// TIA Portal V20 export
// export: Created 2025-12-01T14:57:10.651905Z, ExportSetting None, DisplayName Totally Integrated Automation Portal, DisplayVersion V20 Update 3, DisplayName TIA Portal Openness, DisplayVersion V20 Update 3, DisplayName TIA Portal Version Control Interface, DisplayVersion V20 Update 3, DisplayName STEP 7 Professional, DisplayVersion V20 Update 3, DisplayName STEP 7 Safety, DisplayVersion V20 Update 2, DisplayName WinCC Basic/Comfort/Advanced, DisplayVersion V20 Update 3, DisplayName WinCC Professional, DisplayVersion V20 Update 3, DisplayName WinCC Unified, DisplayVersion V20 Update 3
FUNCTION "FC822_EstadosMesas" : Void   // FC822, LAD
TITLE = "EstadosMesas" - Calcular los eventos con las Mesas
{ S7_Optimized_Access := 'FALSE' }
AUTHOR : TRACKING
NAME : 20170706
VERSION : 4.6
// - Inicializaciones
// - Bucle de Mesas
// - Cierre de protocolo
// - Calculo de los Eventos con Presencias
// - Calculo de los Eventos Generales
// stored: AutoNumber false, SetENOAutomatically false
   VAR_TEMP
      EmiProtocoloDeMesa : "UDT_ProtocoloEmiMesa";
      P_EmiProtocolo : DWord;
      NumeroMesa : UInt;   // Numero de Mesa Actual
      NumeroUT : UInt;   // Numero de UT Actual
      SiguienteUT : UInt;   // Numero de UT Siguiente
      AnteriorUT : UInt;
      GaliboTMP : Word;
      HuecoTacoTMP : Word;
      AlturaTMP : UInt;
      ValorTMP : UInt;
      GrupoTMP : UInt;
   END_VAR
BEGIN

NETWORK
TITLE = Inicializar
// - Inicializacion de las variables de los DB's
/////////////////////////////////////////////////////////////////////////
// --- Inicializaciones de las variables de los DB's



NETWORK
TITLE = Bucle de Mesas
// - Inicializacion de los punteros de la mesa (PunteroMesa y PunteroPLC)
// - Inicializacion de la definicion de la Mesa
// - Mirar si ha cerrado el protocolo
// - Mirar si hay UT's en la Mesa
// -
/////////////////////////////////////////////////////////////////////////
//                      Recorrer todas las Mesas
/////////////////////////////////////////////////////////////////////////
// -- Inicializacion de los Punteros de la Mesa
// -- Miarar si ha cerrado el protocolo de la Mesa

      L     0;  // Inicializo variable, para bucle de mesas
      T     #NumeroMesa;

/////////////////////////////////////////////////////////////////////////
// --- Empieza el recorrido por todas las Mesas
InicioBucle_Mesas:NOP   0;
      L     #NumeroMesa;  // Incremento en uno el numero de mesa
      L     1;
      +I;
      T     #NumeroMesa;


/////////////////////////////////////////////////////////////////////////
// Ya estan todas las Mesas
      L     #NumeroMesa;
      L     "CTE_MaxMesas";
      >I;
      JC    _END;  // Ya he recorrido todas las Mesas


/////////////////////////////////////////////////////////////////////////
/// Mirar Si hay Mesa Configurada

      SET;
      AN    "DB850_DefinicionMesas".Mesa[#NumeroMesa].ConfigMesa.MesaPaso;
      AN    "DB850_DefinicionMesas".Mesa[#NumeroMesa].ConfigMesa.MesaCruce;
      AN    "DB850_DefinicionMesas".Mesa[#NumeroMesa].ConfigMesa.MesaMultiplesDestinos;
      AN    "DB850_DefinicionMesas".Mesa[#NumeroMesa].ConfigMesa.MesaTL;
      JC    InicioBucle_Mesas;


/////////////////////////////////////////////////////////////////////////
/// Recoger Datos de Emision y Recepcion
// --- Recoger Datos del Dispositivo (Protocolo)
      CALL  MOVE
      ( IN  := "DB840_Emision".Mesa[#NumeroMesa].Protocolo,
        OUT := #EmiProtocoloDeMesa
      );

      L     P##EmiProtocoloDeMesa;
      T     #P_EmiProtocolo;


/////////////////////////////////////////////////////////////////////////
// --- Mirar si ha cerrado el protocolo de la Mesa

      L     "DB810_ColasMesas".Colas[#NumeroMesa].EstadoPresenciaMesa;
      L     0;  // Mirar si no esta Cerrado el Protocolo
      <>I;  // Ir a Cerrar Protocolo de la Mesa
      JC    CerrarProtocolo_Mesa;


/////////////////////////////////////////////////////////////////////////
// --- Mirar si hay UT's en la Mesa
//     Mirar si existe una UT, coger la primera
      L     "DB810_ColasMesas".Colas[#NumeroMesa].UT_PrimeraMesa;
      T     #NumeroUT;  // UT_Primera

      L     #NumeroUT;
      L     0;
      ==I;
      JC    InicioBucle_Mesas;  // No hay UT's en la Mesa, Siguiente Mesa


/////////////////////////////////////////////////////////////////////////
// --- Tratar la Mesa
      JU    TratarPresencias_Mesa;



NETWORK
TITLE = Cierre del protocolo de la mesa
// - Recoger como esta la Presencia
// - Distribuir dependiendo del Status del Protocolo
//   * Esta en Fase 1 - Esperando que se desactive la Presencia de la Mesa
CerrarProtocolo_Mesa:NOP   0;

/////////////////////////////////////////////////////////////////////////
/////////////////////////////////////////////////////////////////////////
/////////////////////////////////////////////////////////////////////////
/////////////////////////////////////////////////////////////////////////
// --- Mirar si ha desactivado todas las presencias
      L     LW [#P_EmiProtocolo];
      L     W#16#FF7F;
      AW;
      L     0;
      <>I;  // Estan Desactivados ?
      JC    FinCerrarProtocolo_Mesa;


/////////////////////////////////////////////////////////////////////////
// --- Fase 1 - Esperando que se desactive Emision de la Mesa
      SET;  // DesActivar - EmiOK de la Mesa
      R     "DB841_Recepcion".Mesa[#NumeroMesa].Protocolo.EmiOK;

      L     0;  // Fase 0 - Acabado el Protocolo
      T     "DB810_ColasMesas".Colas[#NumeroMesa].EstadoPresenciaMesa;


/////////////////////////////////////////////////////////////////////////
// --- Final del Segmento del Cierre de Protocolo de la Mesa
FinCerrarProtocolo_Mesa:NOP   0;
// Finalizar, Siguiente Mesa
      JU    InicioBucle_Mesas;



NETWORK
TITLE = Empezar el cierre del protocolo
// Empezar el cierre del protocolo - Empezar el EmiOK
EmpezarProtocolo_Mesa:NOP   0;

/////////////////////////////////////////////////////////////////////////
/////////////////////////////////////////////////////////////////////////
/////////////////////////////////////////////////////////////////////////
/////////////////////////////////////////////////////////////////////////
// --- Empezar el cierre del protocolo
      SET;  // Activar - EmiOK de la Mesa
      S     "DB841_Recepcion".Mesa[#NumeroMesa].Protocolo.EmiOK;

      L     1;  // Fase 1, Empezar el Protocolo
      T     "DB810_ColasMesas".Colas[#NumeroMesa].EstadoPresenciaMesa;


/////////////////////////////////////////////////////////////////////////
// Finalizar, Siguiente Mesa
      JU    InicioBucle_Mesas;



NETWORK
TITLE = Tratamiento de la Mesa
// - Tratamiento de la presencia de una mesa
//   * Leer del PLC la Zona de Bits
//   * Miramos si hay alguno activo
//     * Si hay alguno: Distribucion del Tipo de Presencias
//     * Si no hay alguno: Vamos a Generales
TratarPresencias_Mesa:NOP   0;

/////////////////////////////////////////////////////////////////////////
/////////////////////////////////////////////////////////////////////////
/////////////////////////////////////////////////////////////////////////
// --- Miramos si hay alguno activo

      L     LW [#P_EmiProtocolo];  // Zona de Bits
      L     W#16#FF7F;  // Quitamos el bit RecepOK
      AW;
      L     0;  // Mirar si hay alguno activo
      ==I;  // Ir a tratar Estado General
      JC    TratarEstadoGeneral_Mesa;

/////////////////////////////////////////////////////////////////////////
/////////////////////////////////////////////////////////////////////////
// --- Distribuir dependiendo del tipo de presencia

/////////////////////////////////////////////////////////////////////////
// Evento de Presencia Normal
      SET;  // Al final de la Cola
      A     #EmiProtocoloDeMesa.PresNormal;
      AN    #EmiProtocoloDeMesa.PresReset;
      AN    "DB850_DefinicionMesas".Mesa[#NumeroMesa].ConfigMesa.MeterAlPrincipio;
      JC    TratarPresenciaUltimaUT_Mesa;

      SET;  // Al principio de la Cola
      A     #EmiProtocoloDeMesa.PresNormal;
      AN    #EmiProtocoloDeMesa.PresReset;
      A     "DB850_DefinicionMesas".Mesa[#NumeroMesa].ConfigMesa.MeterAlPrincipio;
      JC    TratarPresenciaPrimeraUT_Mesa;

/////////////////////////////////////////////////////////////////////////
// Evento de Presencia con Galibo
      SET;  // Al final de la Cola
      A     #EmiProtocoloDeMesa.PresGalibo;
      AN    "DB850_DefinicionMesas".Mesa[#NumeroMesa].ConfigMesa.MeterAlPrincipio;
      JC    TratarGaliboUltimaUT_Mesa;

      SET;  // Al principio de la Cola
      A     #EmiProtocoloDeMesa.PresGalibo;
      A     "DB850_DefinicionMesas".Mesa[#NumeroMesa].ConfigMesa.MeterAlPrincipio;
      JC    TratarGaliboPrimeraUT_Mesa;

/////////////////////////////////////////////////////////////////////////
// Evento de Presencia con Bloqueo
      SET;
      A     #EmiProtocoloDeMesa.PresBloqueo;
      JC    TratarPresenciaBloqueo_Mesa;

/////////////////////////////////////////////////////////////////////////
// Evento de Presencia de Reset
      SET;
      A     #EmiProtocoloDeMesa.PresNormal;
      A     #EmiProtocoloDeMesa.PresReset;
      JC    TratarPresenciaReset_Mesa;

/////////////////////////////////////////////////////////////////////////
// Evento de Ausencia
      SET;  // (BORRAR UT)
      A     "DB850_DefinicionMesas".Mesa[#NumeroMesa].ConfigMesa.AusenciaBorrarUT;
      A     #EmiProtocoloDeMesa.Ausencia;
      JC    TratarAusenciaBorrar_Mesa;

      SET;  // (NORMAL)
      AN    "DB850_DefinicionMesas".Mesa[#NumeroMesa].ConfigMesa.AusenciaBorrarUT;
      A     #EmiProtocoloDeMesa.Ausencia;
      JC    TratarAusenciaNormal_Mesa;


/////////////////////////////////////////////////////////////////////////
// --- Si llega aqui este tipo no esta programado
// Ir a Empezar el Cierre de Protocolo
      JU    CerrarProtocolo_Mesa;



NETWORK
TITLE = Tratamiento de los Eventos Generales
// - Recorrer todas las UT's de la Mesa
//   - Recoger datos de la UT
//   - Mirar si se pueden generar eventos
//     * StatusEventoAGenerar = 0
//     * StatusEmision = 0
//     * StatusRecepcion = 0
//   - Mirar si tiene eventos generales
//     * Evento de Peticion de ruta 
//     * Evento de Refesco de datos
//     * Evento de Peticion de datos
//     * Nueva UT en Mesa (No se debe dar nunca)
//     * Borrar UT
// - Siguiente UT (Si hay más en la Mesa)
TratarEstadoGeneral_Mesa:NOP   0;

/////////////////////////////////////////////////////////////////////////
/////////////////////////////////////////////////////////////////////////
/////////////////////////////////////////////////////////////////////////
// --- Recorrer todas las Ut's de la Mesa
InicioBucleUTs_Mesa:NOP   0;

/////////////////////////////////////////////////////////////////////////
// --- Mirar si de pueden Generar eventos
//     - Si hay algo para generar
//     - Si puede ?

// --- No hay nada que generar
      L     "DB812_UTs_Control".UT[#NumeroUT].EstadoGeneralUT;
      L     0;  // EstaodGeneralUT <> 0
      ==I;  // Siguiente UT de la Mesa, No hay
      JC    ContinuarBucleUTs_Mesa;

// --- Se puede ?
      L     "DB812_UTs_Control".UT[#NumeroUT].EstadoEventoAGenerar;
      L     0;  // EstaodEventoAGenerar = 0
      <>I;  // Siguiente UT de la Mesa, No se puede
      JC    ContinuarBucleUTs_Mesa;

// --- Siempre se Borra UT
//     Evento de BorrarUT
      L     "DB812_UTs_Control".UT[#NumeroUT].EstadoGeneralUT;
      L     31;  // 31 - Borrar UT
      ==I;  // No hay cumplir las Condiciones
      JC    BorrarUT_EstadoGeneral_Mesa;

// EstaodEmisionUT = 0
      L     "DB812_UTs_Control".UT[#NumeroUT].EstadoEmisionUT;
      L     0;  // EstaodEmisionUT = 0
      <>I;  // Siguiente UT de la Mesa, No se puede
      JC    ContinuarBucleUTs_Mesa;

// EstaodRecepcionUT = 0
      L     "DB812_UTs_Control".UT[#NumeroUT].EstadoRecepcionUT;
      L     0;  // EstaodRecepcionUT = 0
      <>I;
      JC    ContinuarBucleUTs_Mesa;  // Siguiente UT de la Mesa, No se puede


/////////////////////////////////////////////////////////////////////////
/////////////////////////////////////////////////////////////////////////
// --- Distribucion de Eventos Generales
//     - Evento de Peticion de Ruta
//     - Evento de Refresco de Datos
//     - Evento de Peticion de Datos
//     - Evento de Nueva UT en la Mesa (NO SE PUEDE DAR)
//     - Evento de BorrarUT

      L     "DB812_UTs_Control".UT[#NumeroUT].EstadoGeneralUT;
      L     21;  // 21 - Peticion de Ruta Nueva
      ==I;  //      LLEGA A SU DESTINO
      JC    PeticionRuta_EnDestinoUT_EstadoGeneral_Mesa;

      L     "DB812_UTs_Control".UT[#NumeroUT].EstadoGeneralUT;
      L     25;  // 25 - Peticion de Ruta Nueva
      ==I;  //      NO TIENE DESTINO
      JC    PeticionRuta_SinDestinoUT_EstadoGeneral_Mesa;

      L     "DB812_UTs_Control".UT[#NumeroUT].EstadoGeneralUT;
      L     26;  // 26 - Peticion de Ruta Nueva
      ==I;  //      FUERA DE RUTA
      JC    PeticionRuta_FueraDeRutaUT_EstadoGeneral_Mesa;


      L     "DB812_UTs_Control".UT[#NumeroUT].EstadoGeneralUT;
      L     22;  // 22 - Refresco de Datos
      ==I;
      JC    RefrescoDatosUT_EstadoGeneral_Mesa;

      L     "DB812_UTs_Control".UT[#NumeroUT].EstadoGeneralUT;
      L     23;  // 23 - Peticion de Datos
      ==I;
      JC    PeticionDatosUT_EstadoGeneral_Mesa;


      L     "DB812_UTs_Control".UT[#NumeroUT].EstadoGeneralUT;
      L     24;  // 24 - Nueva UT
      ==I;
      JC    NuevaUT_EstadoGeneral_Mesa;


      L     "DB812_UTs_Control".UT[#NumeroUT].EstadoGeneralUT;
      L     31;  // 31 - Borrar UT
      ==I;
      JC    BorrarUT_EstadoGeneral_Mesa;


/////////////////////////////////////////////////////////////////////////
/////////////////////////////////////////////////////////////////////////
// --- El evento no esta programado

      L     0;  // Darlo por tratado
      T     "DB812_UTs_Control".UT[#NumeroUT].EstadoGeneralUT;


// Siguiente UT de la Mesa
      JU    ContinuarBucleUTs_Mesa;




/////////////////////////////////////////////////////////////////////////
/////////////////////////////////////////////////////////////////////////
/////////////////////////////////////////////////////////////////////////
// --- Evento de Peticion de Ruta Nueva, Por llegada a Destino
PeticionRuta_EnDestinoUT_EstadoGeneral_Mesa:NOP   0;
      L     123;  // 123 - Generar Evento de Peticion de Ruta
      T     "DB812_UTs_Control".UT[#NumeroUT].EstadoEventoAGenerar;
      L     0;  // Darlo por tratado
      T     "DB812_UTs_Control".UT[#NumeroUT].EstadoGeneralUT;


// Siguiente UT de la Mesa
      JU    ContinuarBucleUTs_Mesa;


/////////////////////////////////////////////////////////////////////////
/////////////////////////////////////////////////////////////////////////
/////////////////////////////////////////////////////////////////////////
// --- Evento de Peticion de Ruta Nueva, Sin Destino
PeticionRuta_SinDestinoUT_EstadoGeneral_Mesa:NOP   0;
      L     124;  // 123 - Generar Evento de Peticion de Ruta
      T     "DB812_UTs_Control".UT[#NumeroUT].EstadoEventoAGenerar;
      L     0;  // Darlo por tratado
      T     "DB812_UTs_Control".UT[#NumeroUT].EstadoGeneralUT;


// Siguiente UT de la Mesa
      JU    ContinuarBucleUTs_Mesa;


/////////////////////////////////////////////////////////////////////////
/////////////////////////////////////////////////////////////////////////
/////////////////////////////////////////////////////////////////////////
// --- Evento de Peticion de Ruta Nueva, Fuera de Ruta
PeticionRuta_FueraDeRutaUT_EstadoGeneral_Mesa:NOP   0;
      L     125;  // 123 - Generar Evento de Peticion de Ruta
      T     "DB812_UTs_Control".UT[#NumeroUT].EstadoEventoAGenerar;
      L     0;  // Darlo por tratado
      T     "DB812_UTs_Control".UT[#NumeroUT].EstadoGeneralUT;


// Siguiente UT de la Mesa
      JU    ContinuarBucleUTs_Mesa;


/////////////////////////////////////////////////////////////////////////
/////////////////////////////////////////////////////////////////////////
/////////////////////////////////////////////////////////////////////////
// --- Evento de Refresco de Datos
RefrescoDatosUT_EstadoGeneral_Mesa:NOP   0;
      L     110;  // 110 - Generar Evento de Refresco de Datos
      T     "DB812_UTs_Control".UT[#NumeroUT].EstadoEventoAGenerar;
      L     0;  // Darlo por tratado
      T     "DB812_UTs_Control".UT[#NumeroUT].EstadoGeneralUT;


// Siguiente UT de la Mesa
      JU    ContinuarBucleUTs_Mesa;


/////////////////////////////////////////////////////////////////////////
/////////////////////////////////////////////////////////////////////////
/////////////////////////////////////////////////////////////////////////
// --- Evento de Peticion de Datos
PeticionDatosUT_EstadoGeneral_Mesa:NOP   0;
      L     141;  // 141 - Generar Evento de Peticion de Datos
      T     "DB812_UTs_Control".UT[#NumeroUT].EstadoEventoAGenerar;
      L     0;  // Darlo por tratado
      T     "DB812_UTs_Control".UT[#NumeroUT].EstadoGeneralUT;


// Siguiente UT de la Mesa
      JU    ContinuarBucleUTs_Mesa;


/////////////////////////////////////////////////////////////////////////
/////////////////////////////////////////////////////////////////////////
/////////////////////////////////////////////////////////////////////////
// --- Evento de Nueva UT (NO SE PUEDE DAR)
NuevaUT_EstadoGeneral_Mesa:NOP   0;
      L     132;  // 132 - Generar Evento de Nueva UT
      L     0;
      T     "DB812_UTs_Control".UT[#NumeroUT].EstadoEventoAGenerar;

      L     0;  // Darlo por tratado
      L     24;
      T     "DB812_UTs_Control".UT[#NumeroUT].EstadoGeneralUT;


// Siguiente UT de la Mesa
      JU    ContinuarBucleUTs_Mesa;


/////////////////////////////////////////////////////////////////////////
/////////////////////////////////////////////////////////////////////////
/////////////////////////////////////////////////////////////////////////
// --- Evento de Borrar UT
BorrarUT_EstadoGeneral_Mesa:NOP   0;
      L     131;  // 131 - Generar Evento de Borrar UT
      T     "DB812_UTs_Control".UT[#NumeroUT].EstadoEventoAGenerar;
      L     0;  // Darlo por tratado
      T     "DB812_UTs_Control".UT[#NumeroUT].EstadoGeneralUT;


// Siguiente UT de la Mesa
      JU    ContinuarBucleUTs_Mesa;




/////////////////////////////////////////////////////////////////////////
/////////////////////////////////////////////////////////////////////////
/////////////////////////////////////////////////////////////////////////
// --- Siguiente UT ? (Mirar si es final de la Mesa)
ContinuarBucleUTs_Mesa:NOP   0;
      L     "DB812_UTs_Control".UT[#NumeroUT].UT_SiguienteMesa;
      T     #SiguienteUT;

      L     #SiguienteUT;
      L     0;  // UT_Siguiente es 0
      ==I;
      JC    FinEstadoGeneral_Mesa;  // Es la Ultima ?

// Siguinete UT
      L     #SiguienteUT;
      T     #NumeroUT;
      JU    InicioBucleUTs_Mesa;



/////////////////////////////////////////////////////////////////////////
/////////////////////////////////////////////////////////////////////////
/////////////////////////////////////////////////////////////////////////
// No hay mas UT's en la mesa --> Se Acabo, Siguiente Mesa
FinEstadoGeneral_Mesa:NOP   0;
      JU    InicioBucle_Mesas;



NETWORK
TITLE = Tratamiento de Presencia Normal Ultima UT
// - Ir a la Ultima UT de la Mesa
//   * Recoger datos de la UT
//   * Condiciones para tratarla
//   * EstadoEmision Correcto
//     * 11 - Cambiado de Mesa
//     * 12 - Nueva UT en la Mesa
TratarPresenciaUltimaUT_Mesa:NOP   0;

/////////////////////////////////////////////////////////////////////////
/////////////////////////////////////////////////////////////////////////
/////////////////////////////////////////////////////////////////////////
// Tratamiento de la Presencia Normal - Ultima UT de la Mesa

InicioBuclePresenciaUltimaUT_Mesa:NOP   0;

// Miramos si es la Ultima UT
      L     "DB812_UTs_Control".UT[#NumeroUT].UT_SiguienteMesa;
      T     #SiguienteUT;

      L     #SiguienteUT;
      L     0;  // UT Siguiente es 0
      ==I;  // ¿Es la Ultima?
      JC    PresenciaUltimaUT_Mesa;

// Si Hay multiples entrada se van validando de camino
      SET;  // Puede haber Multiples Entradas ?
      A     "DB850_DefinicionMesas".Mesa[#NumeroMesa].ConfigMesa.MultiplesCargasDeEntrada;
      O     "DB850_DefinicionMesas".Mesa[#NumeroMesa].ConfigMesa.GrupoDeEntrada;
      JC    MultiplesPresenciaUltimaUT_Mesa;

// Continuar hasta llegar a la ultima UT
ContinuarBuclePresenciaUltimaUT_Mesa:NOP   0;
      L     #SiguienteUT;
      T     #NumeroUT;
      JU    InicioBuclePresenciaUltimaUT_Mesa;



NETWORK
TITLE = --- Ultima UT de la Mesa
/////////////////////////////////////////////////////////////////////////
/////////////////////////////////////////////////////////////////////////
/////////////////////////////////////////////////////////////////////////
// ---
// ---                       ULTIMA UT
/////////////////////////////////////////////////////////////////////////
/////////////////////////////////////////////////////////////////////////
/////////////////////////////////////////////////////////////////////////
// --- Ya se ha encontrado la Ultima UT
//     * Recoger datos de la UT
//     * Condiciones de Uso de la Presencia
//       * EstadoRecepcion = 0
//       * EstadoEventosAGenerar = 0
//     * Estado de la Emision Correcto
PresenciaUltimaUT_Mesa:NOP   0;

/////////////////////////////////////////////////////////////////////////
// --- Condiciones de Uso de la Presencia

      L     "DB812_UTs_Control".UT[#NumeroUT].EstadoEventoAGenerar;
      L     0;  // Esta libre
      <>I;  // No se puede hacer nada todavia
      JC    InicioBucle_Mesas;

      L     "DB812_UTs_Control".UT[#NumeroUT].EstadoRecepcionUT;
      L     0;  // Esta libre
      <>I;  // No se puede hacer nada todavia
      JC    InicioBucle_Mesas;


/////////////////////////////////////////////////////////////////////////
// --- Estado de la Emision Correto

      L     "DB812_UTs_Control".UT[#NumeroUT].EstadoEmisionUT;
      L     11;  // Solo en estado 11 (Cambio de Mesa)
      ==I;  // Ir a generar evento
      JC    CambioDeMesa_PresenciaUltimaUT_Mesa;

      L     "DB812_UTs_Control".UT[#NumeroUT].EstadoEmisionUT;
      L     12;  // Solo en estado 12 (Nueva Paleta)
      ==I;  // Ir a generar evento
      JC    NuevaEnMesa_PresenciaUltimaUT_Mesa;


/////////////////////////////////////////////////////////////////////////
// --- Todavia no se cumple el Estado de Emision correcto
//     No se ha tratado la Presencia
      JU    InicioBucle_Mesas;




/////////////////////////////////////////////////////////////////////////
/////////////////////////////////////////////////////////////////////////
/////////////////////////////////////////////////////////////////////////
// --- (11)- La UT ha cambiado de Mesa
//           * Generar evento
//           * Avisar al generador de ordenes
//           * Dar por tratado la Presencia Normal
CambioDeMesa_PresenciaUltimaUT_Mesa:NOP   0;
      L     11;  // 11 - Cambio de Mesa de la UT
      T     "DB812_UTs_Control".UT[#NumeroUT].EstadoRecepcionUT;
      L     0;  // Darlo por tratado
      T     "DB812_UTs_Control".UT[#NumeroUT].EstadoEmisionUT;

      SET;  // Se debe informar al Jefe de Trafico
      A     "DB850_DefinicionMesas".Mesa[#NumeroMesa].ConfigMesa.NoInformar;
      JC    NoInformarCambioDeMesa_PresenciaUltimaUT_Mesa;

      L     100;  // 100 - Generar Evento de Presencia
      T     "DB812_UTs_Control".UT[#NumeroUT].EstadoEventoAGenerar;

NoInformarCambioDeMesa_PresenciaUltimaUT_Mesa:NOP   0;


/////////////////////////////////////////////////////////////////////////
// ----- Mirar si hay que pedir ruta: .....
      L     "DB812_UTs_Control".UT[#NumeroUT].MesaDestino;
      L     0;  // MesaDestino = 0
      ==I;  // No tiene ruta ?
      JC    CambioDeMesa_SinDestino_PresenciaUltimaUT_Mesa;

      L     "DB812_UTs_Control".UT[#NumeroUT].MesaActual;
      L     "DB812_UTs_Control".UT[#NumeroUT].MesaDestino;  // MesaActual = MesaDestino
      ==I;  // Ha finalizado la ruta ?
      JC    CambioDeMesa_EnDestino_PresenciaUltimaUT_Mesa;


/////////////////////////////////////////////////////////////////////////
// Todavia tiene ruta
      JU    EmpezarProtocolo_Mesa;



/////////////////////////////////////////////////////////////////////////
/////////////////////////////////////////////////////////////////////////
// ---- Pedir ruta: ...... En Destino
CambioDeMesa_EnDestino_PresenciaUltimaUT_Mesa:NOP   0;
      L     21;  // 21 - Genearar Evento Pedir Ruta
      T     "DB812_UTs_Control".UT[#NumeroUT].EstadoGeneralUT;
      L     0;  // Dar por tratada
      T     "DB812_UTs_Control".UT[#NumeroUT].EstadoRecepcionUT;

      JU    EmpezarProtocolo_Mesa;


/////////////////////////////////////////////////////////////////////////
/////////////////////////////////////////////////////////////////////////
// ---- Pedir ruta: ...... Sin destino
CambioDeMesa_SinDestino_PresenciaUltimaUT_Mesa:NOP   0;
      L     25;  // 25 - Generar Evento Pedir Ruta (SIN DESTINO)
      T     "DB812_UTs_Control".UT[#NumeroUT].EstadoGeneralUT;
      L     0;  // Dar por tratada
      T     "DB812_UTs_Control".UT[#NumeroUT].EstadoRecepcionUT;

      JU    EmpezarProtocolo_Mesa;




/////////////////////////////////////////////////////////////////////////
/////////////////////////////////////////////////////////////////////////
/////////////////////////////////////////////////////////////////////////
// --- (12)- Nueva UT en Mesa
//           * Generar evento
//           * Avisar al generador de ordenes
//           * Dar por tratado la Presencia Normal
NuevaEnMesa_PresenciaUltimaUT_Mesa:NOP   0;
      L     12;  // 12 - Nueva UT en Mesa
      T     "DB812_UTs_Control".UT[#NumeroUT].EstadoRecepcionUT;
      L     0;  // Darlo por tratado
      T     "DB812_UTs_Control".UT[#NumeroUT].EstadoEmisionUT;

      L     132;  // 132 - Generar Evento de Nueva UT
      T     "DB812_UTs_Control".UT[#NumeroUT].EstadoEventoAGenerar;

      JU    EmpezarProtocolo_Mesa;



NETWORK
TITLE = --- Resto de UTs de la Mesa (Multiples) - Ultima
/////////////////////////////////////////////////////////////////////////
/////////////////////////////////////////////////////////////////////////
/////////////////////////////////////////////////////////////////////////
//               MULTIPLES ENTRADAS - NO ULTIMA UT
/////////////////////////////////////////////////////////////////////////
/////////////////////////////////////////////////////////////////////////
/////////////////////////////////////////////////////////////////////////
// --- Ya e ha encontrado la alguna UT (Multiples Entradas) y no la Ultima
//     * Recoger datos de la UT
//     * Condiciones Ninguna, solo a la ultima
//     * Estado de la Emision Correcto
MultiplesPresenciaUltimaUT_Mesa:NOP   0;

// --- Condiciones : No necesita nada más que la ultima
// --- Estado de la Emision Correto

      L     "DB812_UTs_Control".UT[#NumeroUT].EstadoEmisionUT;
      L     11;  // Solo en estado 11 (Cambio de Mesa)
      ==I;  // Ir a generar evento
      JC    CambioDeMesa_MultiplesPresenciaUltimaUT_Mesa;

      L     "DB812_UTs_Control".UT[#NumeroUT].EstadoEmisionUT;
      L     12;  // Solo en estado 12 (Nueva Carga)
      ==I;  // Ir a generar evento
      JC    NuevaEnMesa_MultiplesPresenciaUltimaUT_Mesa;

// No necesita, continuar buscando la Ultima UT
      JU    ContinuarBuclePresenciaUltimaUT_Mesa;



/////////////////////////////////////////////////////////////////////////
/////////////////////////////////////////////////////////////////////////
/////////////////////////////////////////////////////////////////////////
// --- (11)- La UT ha cambiado de Mesa
//           * Generar evento
//           * Mirar si hay que pedir ruta
//           * Avisar al generador de ordenes
CambioDeMesa_MultiplesPresenciaUltimaUT_Mesa:NOP   0;
      L     11;  // 11 - Cambio de Mesa de la UT
      T     "DB812_UTs_Control".UT[#NumeroUT].EstadoRecepcionUT;
      L     0;  // Darlo por tratado
      T     "DB812_UTs_Control".UT[#NumeroUT].EstadoEmisionUT;

      SET;  // Se debe informar al Jefe de Trafico
      A     "DB850_DefinicionMesas".Mesa[#NumeroMesa].ConfigMesa.NoInformar;
      JC    NoInformarCambioDeMesa_MultiplesPresenciaUltimaUT_Mesa;

      L     100;  // 100 - Generar Evento de Presencia
      T     "DB812_UTs_Control".UT[#NumeroUT].EstadoEventoAGenerar;

NoInformarCambioDeMesa_MultiplesPresenciaUltimaUT_Mesa:NOP   0;


/////////////////////////////////////////////////////////////////////////
// ----- Mirar si hay que pedir ruta: .....
      L     "DB812_UTs_Control".UT[#NumeroUT].MesaDestino;
      L     0;  // MesaDestino = 0
      ==I;  // No tiene ruta ?
      JC    CambioDeMesa_SinDestino_MultiplesPresenciaUltimaUT_Mesa;

      L     "DB812_UTs_Control".UT[#NumeroUT].MesaDestino;
      L     "DB812_UTs_Control".UT[#NumeroUT].MesaActual;  // MesaActual = MesaDestino
      ==I;  // Ha finalizado la ruta ?
      JC    CambioDeMesa_EnDestino_MultiplesPresenciaUltimaUT_Mesa;


/////////////////////////////////////////////////////////////////////////
// Todavia tiene ruta
      JU    ContinuarBuclePresenciaUltimaUT_Mesa;


/////////////////////////////////////////////////////////////////////////
/////////////////////////////////////////////////////////////////////////
// ---- Pedir ruta: ...... En Destino
CambioDeMesa_EnDestino_MultiplesPresenciaUltimaUT_Mesa:NOP   0;
      L     21;  // 21 - Generar Evento Pedir Ruta
      T     "DB812_UTs_Control".UT[#NumeroUT].EstadoGeneralUT;
      L     0;  // Dar por tratada
      T     "DB812_UTs_Control".UT[#NumeroUT].EstadoRecepcionUT;

      JU    ContinuarBuclePresenciaUltimaUT_Mesa;


/////////////////////////////////////////////////////////////////////////
/////////////////////////////////////////////////////////////////////////
// ---- Pedir ruta: ...... Sin Destino
CambioDeMesa_SinDestino_MultiplesPresenciaUltimaUT_Mesa:NOP   0;
      L     25;  // 25 - Generar Evento Pedir Ruta (NO DESTINO)
      T     "DB812_UTs_Control".UT[#NumeroUT].EstadoGeneralUT;
      L     0;  // Dar por tratada
      T     "DB812_UTs_Control".UT[#NumeroUT].EstadoRecepcionUT;

      JU    ContinuarBuclePresenciaUltimaUT_Mesa;



/////////////////////////////////////////////////////////////////////////
/////////////////////////////////////////////////////////////////////////
/////////////////////////////////////////////////////////////////////////
// --- (12)- Nueva UT en Mesa
//           * Generar evento
//           * Avisar al generador de ordenes
NuevaEnMesa_MultiplesPresenciaUltimaUT_Mesa:NOP   0;
      L     12;  // 12 - Nueva UT en Mesa
      T     "DB812_UTs_Control".UT[#NumeroUT].EstadoRecepcionUT;
      L     0;  // Darlo por tratado
      T     "DB812_UTs_Control".UT[#NumeroUT].EstadoEmisionUT;

      L     132;  // 132 - Generar Evento de Nueva UT
      T     "DB812_UTs_Control".UT[#NumeroUT].EstadoEventoAGenerar;

      JU    ContinuarBuclePresenciaUltimaUT_Mesa;



NETWORK
TITLE = Tratamiento de Presencia Normal Primera UT
// - Ir a la Primera UT de la Mesa (Pero Recorriendo al Reves)
//   * Recoger datos de la UT
//   * Condiciones para tratarla
//   * EstadoEmision Correcto
//     * 11 - Cambiado de Mesa
//     * 12 - Nueva UT en la Mesa
TratarPresenciaPrimeraUT_Mesa:NOP   0;

/////////////////////////////////////////////////////////////////////////
/////////////////////////////////////////////////////////////////////////
/////////////////////////////////////////////////////////////////////////
// Tratamiento de la Presencia Normal - Pimera UT de la Mesa

/////////////////////////////////////////////////////////////////////////
// --- Realizar el tramiento al Reves --- Buscar la ultima UT primero
BucleBuscarUltimaUT_PresenciaPrimeraUT_Mesa:NOP   0;

      L     "DB812_UTs_Control".UT[#NumeroUT].UT_SiguienteMesa;
      T     #SiguienteUT;

      L     #SiguienteUT;
      L     0;  // UT Siguiente es 0
      ==I;  // ¿Es la Ultima?
      JC    EncontradaUltimaUT_PresenciaPrimeraUT_Mesa;

      L     #SiguienteUT;
      T     #NumeroUT;
      JU    BucleBuscarUltimaUT_PresenciaPrimeraUT_Mesa;

// --- Ya econtrada la Ultima, descendemos
EncontradaUltimaUT_PresenciaPrimeraUT_Mesa:NOP   0;


/////////////////////////////////////////////////////////////////////////
// --- Recorremos la Mesa pero buscando la primera UT
InicioBuclePresenciaPrimeraUT_Mesa:NOP   0;

// --- Miramos si es la Primera UT
      L     "DB812_UTs_Control".UT[#NumeroUT].UT_AnteriorMesa;
      T     #AnteriorUT;

      L     #AnteriorUT;  // ¿Es la Primera?
      L     0;  // UT Siguiente es 0
      ==I;
      JC    PresenciaPrimeraUT_Mesa;  // Es la Primera

// Si Hay multiples entrada se van validando de camino
      SET;
      A     "DB850_DefinicionMesas".Mesa[#NumeroMesa].ConfigMesa.MultiplesCargasDeEntrada;
      O     "DB850_DefinicionMesas".Mesa[#NumeroMesa].ConfigMesa.GrupoDeEntrada;
      JC    MultiplesPresenciaPrimeraUT_Mesa;

// Continuar hasta llegar a la Primera UT
ContinuarBuclePresenciaPrimeraUT_Mesa:NOP   0;
      L     #AnteriorUT;
      T     #NumeroUT;
      JU    InicioBuclePresenciaPrimeraUT_Mesa;



NETWORK
TITLE = --- Primera UT de la Mesa
/////////////////////////////////////////////////////////////////////////
/////////////////////////////////////////////////////////////////////////
/////////////////////////////////////////////////////////////////////////
// ---                       PRIMERA UT
/////////////////////////////////////////////////////////////////////////
/////////////////////////////////////////////////////////////////////////
/////////////////////////////////////////////////////////////////////////
// --- Ya se ha encontrado la Primera UT
//     * Recoger datos de la UT
//     * Condiciones de Uso de la Presencia
//       * EstadoRecepcion = 0
//       * EstadoEventosAGenerar = 0
//     * Estado de la Emision Correcto
PresenciaPrimeraUT_Mesa:NOP   0;

/////////////////////////////////////////////////////////////////////////
// --- Condiciones de Uso de la Presencia

      L     "DB812_UTs_Control".UT[#NumeroUT].EstadoEventoAGenerar;
      L     0;  // Esta libre
      <>I;  // No se puede hacer nada todavia
      JC    InicioBucle_Mesas;

      L     "DB812_UTs_Control".UT[#NumeroUT].EstadoRecepcionUT;
      L     0;  // Esta libre
      <>I;  // No se puede hacer nada todavia
      JC    InicioBucle_Mesas;


/////////////////////////////////////////////////////////////////////////
// --- Estado de la Emision Correto

      L     "DB812_UTs_Control".UT[#NumeroUT].EstadoEmisionUT;
      L     11;  // Solo en estado 11 (Cambio de Mesa)
      ==I;  // Ir a generar evento
      JC    CambioDeMesa_PresenciaPrimeraUT_Mesa;

      L     "DB812_UTs_Control".UT[#NumeroUT].EstadoEmisionUT;
      L     12;  // Solo en estado 12 (Nueva Paleta)
      ==I;  // Ir a generar evento
      JC    NuevaEnMesa_PresenciaPrimeraUT_Mesa;


/////////////////////////////////////////////////////////////////////////
// --- Todavia no se cumple el Estado de Emision correcto
//     No se ha tratado la Presencia
      JU    InicioBucle_Mesas;




/////////////////////////////////////////////////////////////////////////
/////////////////////////////////////////////////////////////////////////
/////////////////////////////////////////////////////////////////////////
// --- (11)- La UT ha cambiado de Mesa
//           * Generar evento
//           * Avisar al generador de ordenes
//           * Dar por tratado la Presencia Normal
CambioDeMesa_PresenciaPrimeraUT_Mesa:NOP   0;
      L     11;  // 11 - Cambio de Mesa de la UT
      T     "DB812_UTs_Control".UT[#NumeroUT].EstadoRecepcionUT;
      L     0;  // Darlo por tratado
      T     "DB812_UTs_Control".UT[#NumeroUT].EstadoEmisionUT;

      SET;  // Se debe informar al Jefe de Trafico
      A     "DB850_DefinicionMesas".Mesa[#NumeroMesa].ConfigMesa.NoInformar;
      JC    NoInformarCambioDeMesa_PresenciaPrimeraUT_Mesa;

      L     100;  // 100 - Generar Evento de Presencia
      T     "DB812_UTs_Control".UT[#NumeroUT].EstadoEventoAGenerar;

NoInformarCambioDeMesa_PresenciaPrimeraUT_Mesa:NOP   0;


/////////////////////////////////////////////////////////////////////////
// ----- Mirar si hay que pedir ruta: .....
      L     "DB812_UTs_Control".UT[#NumeroUT].MesaDestino;
      L     0;  // MesaDestino = 0
      ==I;  // No tiene ruta ?
      JC    CambioDeMesa_SinDestino_PresenciaPrimeraUT_Mesa;

      L     "DB812_UTs_Control".UT[#NumeroUT].MesaActual;
      L     "DB812_UTs_Control".UT[#NumeroUT].MesaDestino;  // MesaActual = MesaDestino
      ==I;  // Ha finalizado la ruta ?
      JC    CambioDeMesa_EnDestino_PresenciaPrimeraUT_Mesa;


/////////////////////////////////////////////////////////////////////////
// Todavia tiene ruta
      JU    EmpezarProtocolo_Mesa;


/////////////////////////////////////////////////////////////////////////
/////////////////////////////////////////////////////////////////////////
// ---- Pedir ruta: ...... En Destino
CambioDeMesa_EnDestino_PresenciaPrimeraUT_Mesa:NOP   0;
      L     21;  // 21 - Genearar Evento Pedir Ruta
      T     "DB812_UTs_Control".UT[#NumeroUT].EstadoGeneralUT;
      L     0;  // Dar por tratada
      T     "DB812_UTs_Control".UT[#NumeroUT].EstadoRecepcionUT;

      JU    EmpezarProtocolo_Mesa;


/////////////////////////////////////////////////////////////////////////
/////////////////////////////////////////////////////////////////////////
// ---- Pedir ruta: ...... Sin destino
CambioDeMesa_SinDestino_PresenciaPrimeraUT_Mesa:NOP   0;
      L     25;  // 25 - Generar Evento Pedir Ruta (SIN DESTINO)
      T     "DB812_UTs_Control".UT[#NumeroUT].EstadoGeneralUT;
      L     0;  // Dar por tratada
      T     "DB812_UTs_Control".UT[#NumeroUT].EstadoRecepcionUT;

      JU    EmpezarProtocolo_Mesa;



/////////////////////////////////////////////////////////////////////////
/////////////////////////////////////////////////////////////////////////
/////////////////////////////////////////////////////////////////////////
// --- (12)- Nueva UT en Mesa
//           * Generar evento
//           * Avisar al generador de ordenes
//           * Dar por tratado la Presencia Normal
NuevaEnMesa_PresenciaPrimeraUT_Mesa:NOP   0;
      L     12;  // 12 - Nueva UT en Mesa
      T     "DB812_UTs_Control".UT[#NumeroUT].EstadoRecepcionUT;
      L     0;  // Darlo por tratado
      T     "DB812_UTs_Control".UT[#NumeroUT].EstadoEmisionUT;

      L     132;  // 132 - Generar Evento de Nueva UT
      T     "DB812_UTs_Control".UT[#NumeroUT].EstadoEventoAGenerar;

      JU    EmpezarProtocolo_Mesa;



NETWORK
TITLE = --- Resto de UTs de la Mesa (Multiples) - Primera
/////////////////////////////////////////////////////////////////////////
/////////////////////////////////////////////////////////////////////////
/////////////////////////////////////////////////////////////////////////
// ---                    MULTIPLES ENTRADAS - NO PRIMERA UT
/////////////////////////////////////////////////////////////////////////
/////////////////////////////////////////////////////////////////////////
/////////////////////////////////////////////////////////////////////////
// --- Ya e ha encontrado la alguna UT (Multiples Entradas) y no la primera
//     * Recoger datos de la UT
//     * Condiciones Ninguna, solo a la primera
//     * Estado de la Emision Correcto
MultiplesPresenciaPrimeraUT_Mesa:NOP   0;

// --- Condiciones : No necesita nada más que la ultima
// --- Estado de la Emision Correto

      L     "DB812_UTs_Control".UT[#NumeroUT].EstadoEmisionUT;
      L     11;  // Solo en estado 11 (Cambio de Mesa)
      ==I;  // Ir a generar evento
      JC    CambioDeMesa_MultiplesPresenciaPrimeraUT_Mesa;

      L     "DB812_UTs_Control".UT[#NumeroUT].EstadoEmisionUT;
      L     12;  // Solo en estado 12 (Nueva Carga)
      ==I;  // Ir a generar evento
      JC    NuevaEnMesa_MultiplesPresenciaPrimeraUT_Mesa;

// No necesita, continuar buscando la Ultima UT
      JU    ContinuarBuclePresenciaPrimeraUT_Mesa;



/////////////////////////////////////////////////////////////////////////
/////////////////////////////////////////////////////////////////////////
/////////////////////////////////////////////////////////////////////////
// --- (11)- La UT ha cambiado de Mesa
//           * Generar evento
//           * Mirar si hay que pedir ruta
//           * Avisar al generador de ordenes
CambioDeMesa_MultiplesPresenciaPrimeraUT_Mesa:NOP   0;
      L     11;  // 11 - Cambio de Mesa de la UT
      T     "DB812_UTs_Control".UT[#NumeroUT].EstadoRecepcionUT;
      L     0;  // Darlo por tratado
      T     "DB812_UTs_Control".UT[#NumeroUT].EstadoEmisionUT;

      SET;  // Se debe informar al Jefe de Trafico
      A     "DB850_DefinicionMesas".Mesa[#NumeroMesa].ConfigMesa.NoInformar;
      JC    NoInformarCambioDeMesa_MultiplesPresenciaPrimeraUT_Mesa;

      L     100;  // 100 - Generar Evento de Presencia
      T     "DB812_UTs_Control".UT[#NumeroUT].EstadoEventoAGenerar;

NoInformarCambioDeMesa_MultiplesPresenciaPrimeraUT_Mesa:NOP   0;


/////////////////////////////////////////////////////////////////////////
// ----- Mirar si hay que pedir ruta: .....
      L     "DB812_UTs_Control".UT[#NumeroUT].MesaDestino;
      L     0;  // MesaDestino = 0
      ==I;  // No tiene ruta ?
      JC    CambioDeMesa_SinDestino_MultiplesPresenciaPrimeraUT_Mesa;

      L     "DB812_UTs_Control".UT[#NumeroUT].MesaDestino;
      L     "DB812_UTs_Control".UT[#NumeroUT].MesaActual;  // MesaActual = MesaDestino
      ==I;  // Ha finalizado la ruta ?
      JC    CambioDeMesa_EnDestino_MultiplesPresenciaPrimeraUT_Mesa;


/////////////////////////////////////////////////////////////////////////
// Todavia tiene ruta
      JU    ContinuarBuclePresenciaPrimeraUT_Mesa;


/////////////////////////////////////////////////////////////////////////
/////////////////////////////////////////////////////////////////////////
// ---- Pedir ruta: ...... En Destino
CambioDeMesa_EnDestino_MultiplesPresenciaPrimeraUT_Mesa:NOP   0;
      L     21;  // 21 - Generar Evento Pedir Ruta
      T     "DB812_UTs_Control".UT[#NumeroUT].EstadoGeneralUT;
      L     0;  // Dar por tratada
      T     "DB812_UTs_Control".UT[#NumeroUT].EstadoRecepcionUT;

      JU    ContinuarBuclePresenciaPrimeraUT_Mesa;


/////////////////////////////////////////////////////////////////////////
/////////////////////////////////////////////////////////////////////////
// ---- Pedir ruta: ...... Sin Destino
CambioDeMesa_SinDestino_MultiplesPresenciaPrimeraUT_Mesa:NOP   0;
      L     25;  // 25 - Generar Evento Pedir Ruta (NO DESTINO)
      T     "DB812_UTs_Control".UT[#NumeroUT].EstadoGeneralUT;
      L     0;  // Dar por tratada
      T     "DB812_UTs_Control".UT[#NumeroUT].EstadoRecepcionUT;

      JU    ContinuarBuclePresenciaPrimeraUT_Mesa;



/////////////////////////////////////////////////////////////////////////
/////////////////////////////////////////////////////////////////////////
/////////////////////////////////////////////////////////////////////////
// --- (12)- Nueva UT en Mesa
//           * Generar evento
//           * Avisar al generador de ordenes
NuevaEnMesa_MultiplesPresenciaPrimeraUT_Mesa:NOP   0;
      L     12;  // 12 - Nueva UT en Mesa
      T     "DB812_UTs_Control".UT[#NumeroUT].EstadoRecepcionUT;
      L     0;  // Darlo por tratado
      T     "DB812_UTs_Control".UT[#NumeroUT].EstadoEmisionUT;

      L     132;  // 132 - Generar Evento de Nueva UT
      T     "DB812_UTs_Control".UT[#NumeroUT].EstadoEventoAGenerar;

      JU    ContinuarBuclePresenciaPrimeraUT_Mesa;



NETWORK
TITLE = Tratamiento de Presencia Galibo Ultima UT
// - Ir a la Ultima UT de la Mesa
//   * Recoger datos de la UT
//   * Condiciones para tratarla
//   * EstadoEmision Correcto
//     * 11 - Cambiado de Mesa
//     * 12 - Nueva UT en la Mesa
TratarGaliboUltimaUT_Mesa:NOP   0;

/////////////////////////////////////////////////////////////////////////
/////////////////////////////////////////////////////////////////////////
/////////////////////////////////////////////////////////////////////////
// Tratamiento de la Presencia Normal - Ultima UT de la Mesa

InicioBucleGaliboUltimaUT_Mesa:NOP   0;

// Miramos si es la Ultima UT
      L     "DB812_UTs_Control".UT[#NumeroUT].UT_SiguienteMesa;
      T     #SiguienteUT;

      L     #SiguienteUT;
      L     0;  // UT Siguiente es 0
      ==I;  // ¿Es la Ultima?
      JC    GaliboUltimaUT_Mesa;

// Si Hay multiples entrada se van validando de camino
      SET;  // Puede haber Multiples Entradas ?
      A     "DB850_DefinicionMesas".Mesa[#NumeroMesa].ConfigMesa.MultiplesCargasDeEntrada;
      O     "DB850_DefinicionMesas".Mesa[#NumeroMesa].ConfigMesa.GrupoDeEntrada;
      JC    MultiplesGaliboUltimaUT_Mesa;

// Continuar hasta llegar a la ultima UT
ContinuarBucleGaliboUltimaUT_Mesa:NOP   0;
      L     #SiguienteUT;
      T     #NumeroUT;
      JU    InicioBucleGaliboUltimaUT_Mesa;



NETWORK
TITLE = --- Ultima UT de la Mesa
/////////////////////////////////////////////////////////////////////////
/////////////////////////////////////////////////////////////////////////
/////////////////////////////////////////////////////////////////////////
// ---
// ---                       ULTIMA UT
/////////////////////////////////////////////////////////////////////////
/////////////////////////////////////////////////////////////////////////
/////////////////////////////////////////////////////////////////////////
// --- Ya se ha encontrado la Ultima UT
//     * Recoger datos de la UT
//     * Condiciones de Uso de la Presencia
//       * EstadoRecepcion = 0
//       * EstadoEventosAGenerar = 0
//     * Estado de la Emision Correcto
GaliboUltimaUT_Mesa:NOP   0;

/////////////////////////////////////////////////////////////////////////
// --- Condiciones de Uso de la Presencia

      L     "DB812_UTs_Control".UT[#NumeroUT].EstadoEventoAGenerar;
      L     0;  // Esta libre
      <>I;  // No se puede hacer nada todavia
      JC    InicioBucle_Mesas;

      L     "DB812_UTs_Control".UT[#NumeroUT].EstadoRecepcionUT;
      L     0;  // Esta libre
      <>I;  // No se puede hacer nada todavia
      JC    InicioBucle_Mesas;


/////////////////////////////////////////////////////////////////////////
// --- Estado de la Emision Correto

      L     "DB812_UTs_Control".UT[#NumeroUT].EstadoEmisionUT;
      L     11;  // Solo en estado 11 (Cambio de Mesa)
      ==I;  // Ir a generar evento
      JC    CambioDeMesa_GaliboUltimaUT_Mesa;

      L     "DB812_UTs_Control".UT[#NumeroUT].EstadoEmisionUT;
      L     12;  // Solo en estado 12 (Nueva Paleta)
      ==I;  // Ir a generar evento
      JC    NuevaEnMesa_GaliboUltimaUT_Mesa;


/////////////////////////////////////////////////////////////////////////
// --- Todavia no se cumple el Estado de Emision correcto
//     No se ha tratado la Presencia
      JU    InicioBucle_Mesas;




/////////////////////////////////////////////////////////////////////////
/////////////////////////////////////////////////////////////////////////
/////////////////////////////////////////////////////////////////////////
// --- (11)- La UT ha cambiado de Mesa
//           * Generar evento
//           * Avisar al generador de ordenes
//           * Dar por tratado la Presencia Normal
CambioDeMesa_GaliboUltimaUT_Mesa:NOP   0;
      L     11;  // 11 - Cambio de Mesa de la UT
      T     "DB812_UTs_Control".UT[#NumeroUT].EstadoRecepcionUT;
      L     0;  // Darlo por tratado
      T     "DB812_UTs_Control".UT[#NumeroUT].EstadoEmisionUT;

      SET;  // Se debe informar al Jefe de Trafico
      A     "DB850_DefinicionMesas".Mesa[#NumeroMesa].ConfigMesa.NoInformar;
      JC    NoInformarCambioDeMesa_GaliboUltimaUT_Mesa;

      L     102;  // 102 - Generar Evento de Galibo
      T     "DB812_UTs_Control".UT[#NumeroUT].EstadoEventoAGenerar;

NoInformarCambioDeMesa_GaliboUltimaUT_Mesa:NOP   0;


/////////////////////////////////////////////////////////////////////////
// ----- Mirar si hay que pedir ruta: .....
      L     "DB812_UTs_Control".UT[#NumeroUT].MesaDestino;
      L     0;  // MesaDestino = 0
      ==I;  // No tiene ruta ?
      JC    CambioDeMesa_SinDestino_GaliboUltimaUT_Mesa;

      L     "DB812_UTs_Control".UT[#NumeroUT].MesaActual;
      L     "DB812_UTs_Control".UT[#NumeroUT].MesaDestino;  // MesaActual = MesaDestino
      ==I;  // Ha finalizado la ruta ?
      JC    CambioDeMesa_EnDestino_GaliboUltimaUT_Mesa;


/////////////////////////////////////////////////////////////////////////
// Todavia tiene ruta
      JU    EmpezarProtocolo_Mesa;


/////////////////////////////////////////////////////////////////////////
/////////////////////////////////////////////////////////////////////////
// ---- Pedir ruta: ...... En Destino
CambioDeMesa_EnDestino_GaliboUltimaUT_Mesa:NOP   0;
      L     21;  // 21 - Genearar Evento Pedir Ruta
      T     "DB812_UTs_Control".UT[#NumeroUT].EstadoGeneralUT;
      L     0;  // Dar por tratada
      T     "DB812_UTs_Control".UT[#NumeroUT].EstadoRecepcionUT;

      JU    EmpezarProtocolo_Mesa;


/////////////////////////////////////////////////////////////////////////
/////////////////////////////////////////////////////////////////////////
// ---- Pedir ruta: ...... Sin destino
CambioDeMesa_SinDestino_GaliboUltimaUT_Mesa:NOP   0;
      L     25;  // 25 - Generar Evento Pedir Ruta (SIN DESTINO)
      T     "DB812_UTs_Control".UT[#NumeroUT].EstadoGeneralUT;
      L     0;  // Dar por tratada
      T     "DB812_UTs_Control".UT[#NumeroUT].EstadoRecepcionUT;

      JU    EmpezarProtocolo_Mesa;


/////////////////////////////////////////////////////////////////////////
/////////////////////////////////////////////////////////////////////////
/////////////////////////////////////////////////////////////////////////
// --- (12)- Nueva UT en Mesa
//           * Generar evento
//           * Avisar al generador de ordenes
//           * Dar por tratado la Presencia Normal
NuevaEnMesa_GaliboUltimaUT_Mesa:NOP   0;
      L     12;  // 12 - Nueva UT en Mesa
      T     "DB812_UTs_Control".UT[#NumeroUT].EstadoRecepcionUT;
      L     0;  // Darlo por tratado
      T     "DB812_UTs_Control".UT[#NumeroUT].EstadoEmisionUT;

      L     132;  // 132 - Generar Evento de Nueva UT
      T     "DB812_UTs_Control".UT[#NumeroUT].EstadoEventoAGenerar;

      JU    EmpezarProtocolo_Mesa;



NETWORK
TITLE = --- Resto de UTs de la Mesa (Multiples) - Ultima
/////////////////////////////////////////////////////////////////////////
/////////////////////////////////////////////////////////////////////////
/////////////////////////////////////////////////////////////////////////
//               MULTIPLES ENTRADAS - NO ULTIMA UT
/////////////////////////////////////////////////////////////////////////
/////////////////////////////////////////////////////////////////////////
/////////////////////////////////////////////////////////////////////////
// --- Ya e ha encontrado la alguna UT (Multiples Entradas) y no la Ultima
//     * Recoger datos de la UT
//     * Condiciones Ninguna, solo a la ultima
//     * Estado de la Emision Correcto
MultiplesGaliboUltimaUT_Mesa:NOP   0;

// --- Condiciones : No necesita nada más que la ultima
// --- Estado de la Emision Correto

      L     "DB812_UTs_Control".UT[#NumeroUT].EstadoEmisionUT;
      L     11;  // Solo en estado 11 (Cambio de Mesa)
      ==I;  // Ir a generar evento
      JC    CambioDeMesa_MultiplesGaliboUltimaUT_Mesa;

      L     "DB812_UTs_Control".UT[#NumeroUT].EstadoEmisionUT;
      L     12;  // Solo en estado 12 (Nueva Carga)
      ==I;  // Ir a generar evento
      JC    NuevaEnMesa_MultiplesGaliboUltimaUT_Mesa;

// No necesita, continuar buscando la Ultima UT
      JU    ContinuarBucleGaliboUltimaUT_Mesa;



/////////////////////////////////////////////////////////////////////////
/////////////////////////////////////////////////////////////////////////
/////////////////////////////////////////////////////////////////////////
// --- (11)- La UT ha cambiado de Mesa
//           * Generar evento
//           * Mirar si hay que pedir ruta
//           * Avisar al generador de ordenes
CambioDeMesa_MultiplesGaliboUltimaUT_Mesa:NOP   0;
      L     11;  // 11 - Cambio de Mesa de la UT
      T     "DB812_UTs_Control".UT[#NumeroUT].EstadoRecepcionUT;
      L     0;  // Darlo por tratado
      T     "DB812_UTs_Control".UT[#NumeroUT].EstadoEmisionUT;

      SET;  // Se debe informar al Jefe de Trafico
      A     "DB850_DefinicionMesas".Mesa[#NumeroMesa].ConfigMesa.NoInformar;
      JC    NoInformarCambioDeMesa_MultiplesGaliboUltimaUT_Mesa;

      L     102;  // 102 - Generar Evento de Galibo
      T     "DB812_UTs_Control".UT[#NumeroUT].EstadoEventoAGenerar;

NoInformarCambioDeMesa_MultiplesGaliboUltimaUT_Mesa:NOP   0;


/////////////////////////////////////////////////////////////////////////
// ----- Mirar si hay que pedir ruta: .....
      L     "DB812_UTs_Control".UT[#NumeroUT].MesaDestino;
      L     0;  // MesaDestino = 0
      ==I;  // No tiene ruta ?
      JC    CambioDeMesa_SinDestino_MultiplesGaliboUltimaUT_Mesa;

      L     "DB812_UTs_Control".UT[#NumeroUT].MesaDestino;
      L     "DB812_UTs_Control".UT[#NumeroUT].MesaActual;  // MesaActual = MesaDestino
      ==I;  // Ha finalizado la ruta ?
      JC    CambioDeMesa_EnDestino_MultiplesGaliboUltimaUT_Mesa;


/////////////////////////////////////////////////////////////////////////
// Todavia tiene ruta
      JU    ContinuarBucleGaliboUltimaUT_Mesa;


/////////////////////////////////////////////////////////////////////////
/////////////////////////////////////////////////////////////////////////
// ---- Pedir ruta: ...... En Destino
CambioDeMesa_EnDestino_MultiplesGaliboUltimaUT_Mesa:NOP   0;
      L     21;  // 21 - Generar Evento Pedir Ruta
      T     "DB812_UTs_Control".UT[#NumeroUT].EstadoGeneralUT;
      L     0;  // Dar por tratada
      T     "DB812_UTs_Control".UT[#NumeroUT].EstadoRecepcionUT;

      JU    ContinuarBucleGaliboUltimaUT_Mesa;


/////////////////////////////////////////////////////////////////////////
/////////////////////////////////////////////////////////////////////////
// ---- Pedir ruta: ...... Sin Destino
CambioDeMesa_SinDestino_MultiplesGaliboUltimaUT_Mesa:NOP   0;
      L     25;  // 25 - Generar Evento Pedir Ruta (NO DESTINO)
      T     "DB812_UTs_Control".UT[#NumeroUT].EstadoGeneralUT;
      L     0;  // Dar por tratada
      T     "DB812_UTs_Control".UT[#NumeroUT].EstadoRecepcionUT;

      JU    ContinuarBucleGaliboUltimaUT_Mesa;


/////////////////////////////////////////////////////////////////////////
/////////////////////////////////////////////////////////////////////////
/////////////////////////////////////////////////////////////////////////
// --- (12)- Nueva UT en Mesa
//           * Generar evento
//           * Avisar al generador de ordenes
NuevaEnMesa_MultiplesGaliboUltimaUT_Mesa:NOP   0;
      L     12;  // 12 - Nueva UT en Mesa
      T     "DB812_UTs_Control".UT[#NumeroUT].EstadoRecepcionUT;
      L     0;  // Darlo por tratado
      T     "DB812_UTs_Control".UT[#NumeroUT].EstadoEmisionUT;

      L     132;  // 132 - Generar Evento de Nueva UT
      T     "DB812_UTs_Control".UT[#NumeroUT].EstadoEventoAGenerar;

      JU    ContinuarBucleGaliboUltimaUT_Mesa;



NETWORK
TITLE = Tratamiento de Presencia Galibol Primera UT
// - Ir a la Primera UT de la Mesa (Pero Recorriendo al Reves)
//   * Recoger datos de la UT
//   * Condiciones para tratarla
//   * EstadoEmision Correcto
//     * 11 - Cambiado de Mesa
//     * 12 - Nueva UT en la Mesa
TratarGaliboPrimeraUT_Mesa:NOP   0;

/////////////////////////////////////////////////////////////////////////
/////////////////////////////////////////////////////////////////////////
/////////////////////////////////////////////////////////////////////////
// Tratamiento de la Presencia Normal - Pimera UT de la Mesa

/////////////////////////////////////////////////////////////////////////
// --- Realizar el tramiento al Reves --- Buscar la ultima UT primero
BucleBuscarUltimaUT_GaliboPrimeraUT_Mesa:NOP   0;

      L     "DB812_UTs_Control".UT[#NumeroUT].UT_SiguienteMesa;
      T     #SiguienteUT;

      L     #SiguienteUT;
      L     0;  // UT Siguiente es 0
      ==I;  // ¿Es la Ultima?
      JC    EncontradaUltimaUT_GaliboPrimeraUT_Mesa;

      L     #SiguienteUT;
      T     #NumeroUT;
      JU    BucleBuscarUltimaUT_GaliboPrimeraUT_Mesa;

// --- Ya econtrada la Ultima, descendemos
EncontradaUltimaUT_GaliboPrimeraUT_Mesa:NOP   0;


/////////////////////////////////////////////////////////////////////////
// --- Recorremos la Mesa pero buscando la primera UT
InicioBucleGaliboPrimeraUT_Mesa:NOP   0;

// --- Miramos si es la Primera UT
      L     "DB812_UTs_Control".UT[#NumeroUT].UT_AnteriorMesa;
      T     #AnteriorUT;

      L     #AnteriorUT;  // ¿Es la Primera?
      L     0;  // UT Siguiente es 0
      ==I;
      JC    GaliboPrimeraUT_Mesa;  // Es la Primera

// Si Hay multiples entrada se van validando de camino
      SET;
      A     "DB850_DefinicionMesas".Mesa[#NumeroMesa].ConfigMesa.MultiplesCargasDeEntrada;
      O     "DB850_DefinicionMesas".Mesa[#NumeroMesa].ConfigMesa.GrupoDeEntrada;
      JC    MultiplesGaliboPrimeraUT_Mesa;

// Continuar hasta llegar a la Primera UT
ContinuarBucleGaliboPrimeraUT_Mesa:NOP   0;
      L     #AnteriorUT;
      T     #NumeroUT;
      JU    InicioBucleGaliboPrimeraUT_Mesa;



NETWORK
TITLE = --- Primera UT de la Mesa
/////////////////////////////////////////////////////////////////////////
/////////////////////////////////////////////////////////////////////////
/////////////////////////////////////////////////////////////////////////
// ---                       PRIMERA UT
/////////////////////////////////////////////////////////////////////////
/////////////////////////////////////////////////////////////////////////
/////////////////////////////////////////////////////////////////////////
// --- Ya se ha encontrado la Primera UT
//     * Recoger datos de la UT
//     * Condiciones de Uso de la Presencia
//       * EstadoRecepcion = 0
//       * EstadoEventosAGenerar = 0
//     * Estado de la Emision Correcto
GaliboPrimeraUT_Mesa:NOP   0;

/////////////////////////////////////////////////////////////////////////
// --- Condiciones de Uso de la Presencia

      L     "DB812_UTs_Control".UT[#NumeroUT].EstadoEventoAGenerar;
      L     0;  // Esta libre
      <>I;  // No se puede hacer nada todavia
      JC    InicioBucle_Mesas;

      L     "DB812_UTs_Control".UT[#NumeroUT].EstadoRecepcionUT;
      L     0;  // Esta libre
      <>I;  // No se puede hacer nada todavia
      JC    InicioBucle_Mesas;


/////////////////////////////////////////////////////////////////////////
// --- Estado de la Emision Correto

      L     "DB812_UTs_Control".UT[#NumeroUT].EstadoEmisionUT;
      L     11;  // Solo en estado 11 (Cambio de Mesa)
      ==I;  // Ir a generar evento
      JC    CambioDeMesa_GaliboPrimeraUT_Mesa;

      L     "DB812_UTs_Control".UT[#NumeroUT].EstadoEmisionUT;
      L     12;  // Solo en estado 12 (Nueva Paleta)
      ==I;  // Ir a generar evento
      JC    NuevaEnMesa_GaliboPrimeraUT_Mesa;


/////////////////////////////////////////////////////////////////////////
// --- Todavia no se cumple el Estado de Emision correcto
//     No se ha tratado la Presencia
      JU    InicioBucle_Mesas;




/////////////////////////////////////////////////////////////////////////
/////////////////////////////////////////////////////////////////////////
/////////////////////////////////////////////////////////////////////////
// --- (11)- La UT ha cambiado de Mesa
//           * Generar evento
//           * Avisar al generador de ordenes
//           * Dar por tratado la Presencia Normal
CambioDeMesa_GaliboPrimeraUT_Mesa:NOP   0;
      L     11;  // 11 - Cambio de Mesa de la UT
      T     "DB812_UTs_Control".UT[#NumeroUT].EstadoRecepcionUT;
      L     0;  // Darlo por tratado
      T     "DB812_UTs_Control".UT[#NumeroUT].EstadoEmisionUT;

      SET;  // Se debe informar al Jefe de Trafico
      A     "DB850_DefinicionMesas".Mesa[#NumeroMesa].ConfigMesa.NoInformar;
      JC    NoInformarCambioDeMesa_GaliboPrimeraUT_Mesa;

      L     102;  // 102 - Generar Evento de Galibo
      T     "DB812_UTs_Control".UT[#NumeroUT].EstadoEventoAGenerar;

NoInformarCambioDeMesa_GaliboPrimeraUT_Mesa:NOP   0;


/////////////////////////////////////////////////////////////////////////
// ----- Mirar si hay que pedir ruta: .....
      L     "DB812_UTs_Control".UT[#NumeroUT].MesaDestino;
      L     0;  // MesaDestino = 0
      ==I;  // No tiene ruta ?
      JC    CambioDeMesa_SinDestino_GaliboPrimeraUT_Mesa;

      L     "DB812_UTs_Control".UT[#NumeroUT].MesaActual;
      L     "DB812_UTs_Control".UT[#NumeroUT].MesaDestino;  // MesaActual = MesaDestino
      ==I;  // Ha finalizado la ruta ?
      JC    CambioDeMesa_EnDestino_GaliboPrimeraUT_Mesa;


/////////////////////////////////////////////////////////////////////////
// Todavia tiene ruta
      JU    EmpezarProtocolo_Mesa;


/////////////////////////////////////////////////////////////////////////
/////////////////////////////////////////////////////////////////////////
// ---- Pedir ruta: ...... En Destino
CambioDeMesa_EnDestino_GaliboPrimeraUT_Mesa:NOP   0;
      L     21;  // 21 - Genearar Evento Pedir Ruta
      T     "DB812_UTs_Control".UT[#NumeroUT].EstadoGeneralUT;
      L     0;  // Dar por tratada
      T     "DB812_UTs_Control".UT[#NumeroUT].EstadoRecepcionUT;

      JU    EmpezarProtocolo_Mesa;


/////////////////////////////////////////////////////////////////////////
/////////////////////////////////////////////////////////////////////////
// ---- Pedir ruta: ...... Sin destino
CambioDeMesa_SinDestino_GaliboPrimeraUT_Mesa:NOP   0;
      L     25;  // 25 - Generar Evento Pedir Ruta (SIN DESTINO)
      T     "DB812_UTs_Control".UT[#NumeroUT].EstadoGeneralUT;
      L     0;  // Dar por tratada
      T     "DB812_UTs_Control".UT[#NumeroUT].EstadoRecepcionUT;

      JU    EmpezarProtocolo_Mesa;


/////////////////////////////////////////////////////////////////////////
/////////////////////////////////////////////////////////////////////////
/////////////////////////////////////////////////////////////////////////
// --- (12)- Nueva UT en Mesa
//           * Generar evento
//           * Avisar al generador de ordenes
//           * Dar por tratado la Presencia Normal
NuevaEnMesa_GaliboPrimeraUT_Mesa:NOP   0;
      L     12;  // 12 - Nueva UT en Mesa
      T     "DB812_UTs_Control".UT[#NumeroUT].EstadoRecepcionUT;
      L     0;  // Darlo por tratado
      T     "DB812_UTs_Control".UT[#NumeroUT].EstadoEmisionUT;

      L     132;  // 132 - Generar Evento de Nueva UT
      T     "DB812_UTs_Control".UT[#NumeroUT].EstadoEventoAGenerar;

      JU    EmpezarProtocolo_Mesa;



NETWORK
TITLE = --- Resto de UTs de la Mesa (Multiples) - Primera
/////////////////////////////////////////////////////////////////////////
/////////////////////////////////////////////////////////////////////////
/////////////////////////////////////////////////////////////////////////
// ---                    MULTIPLES ENTRADAS - NO PRIMERA UT
/////////////////////////////////////////////////////////////////////////
/////////////////////////////////////////////////////////////////////////
/////////////////////////////////////////////////////////////////////////
// --- Ya e ha encontrado la alguna UT (Multiples Entradas) y no la primera
//     * Recoger datos de la UT
//     * Condiciones Ninguna, solo a la primera
//     * Estado de la Emision Correcto
MultiplesGaliboPrimeraUT_Mesa:NOP   0;

// --- Condiciones : No necesita nada más que la ultima
// --- Estado de la Emision Correto

      L     "DB812_UTs_Control".UT[#NumeroUT].EstadoEmisionUT;
      L     11;  // Solo en estado 11 (Cambio de Mesa)
      ==I;  // Ir a generar evento
      JC    CambioDeMesa_MultiplesGaliboPrimeraUT_Mesa;

      L     "DB812_UTs_Control".UT[#NumeroUT].EstadoEmisionUT;
      L     12;  // Solo en estado 12 (Nueva Carga)
      ==I;  // Ir a generar evento
      JC    NuevaEnMesa_MultiplesGaliboPrimeraUT_Mesa;

// No necesita, continuar buscando la Ultima UT
      JU    ContinuarBucleGaliboPrimeraUT_Mesa;



/////////////////////////////////////////////////////////////////////////
/////////////////////////////////////////////////////////////////////////
/////////////////////////////////////////////////////////////////////////
// --- (11)- La UT ha cambiado de Mesa
//           * Generar evento
//           * Mirar si hay que pedir ruta
//           * Avisar al generador de ordenes
CambioDeMesa_MultiplesGaliboPrimeraUT_Mesa:NOP   0;
      L     11;  // 11 - Cambio de Mesa de la UT
      T     "DB812_UTs_Control".UT[#NumeroUT].EstadoRecepcionUT;
      L     0;  // Darlo por tratado
      T     "DB812_UTs_Control".UT[#NumeroUT].EstadoEmisionUT;

      SET;  // Se debe informar al Jefe de Trafico
      A     "DB850_DefinicionMesas".Mesa[#NumeroMesa].ConfigMesa.NoInformar;
      JC    NoInformarCambioDeMesa_MultiplesGaliboPrimeraUT_Mesa;

      L     102;  // 102 - Generar Evento de Galibo
      T     "DB812_UTs_Control".UT[#NumeroUT].EstadoEventoAGenerar;

NoInformarCambioDeMesa_MultiplesGaliboPrimeraUT_Mesa:NOP   0;


/////////////////////////////////////////////////////////////////////////
// ----- Mirar si hay que pedir ruta: .....
      L     "DB812_UTs_Control".UT[#NumeroUT].MesaDestino;
      L     0;  // MesaDestino = 0
      ==I;  // No tiene ruta ?
      JC    CambioDeMesa_SinDestino_MultiplesGaliboPrimeraUT_Mesa;

      L     "DB812_UTs_Control".UT[#NumeroUT].MesaDestino;
      L     "DB812_UTs_Control".UT[#NumeroUT].MesaActual;  // MesaActual = MesaDestino
      ==I;  // Ha finalizado la ruta ?
      JC    CambioDeMesa_EnDestino_MultiplesGaliboPrimeraUT_Mesa;


/////////////////////////////////////////////////////////////////////////
// Todavia tiene ruta
      JU    ContinuarBucleGaliboPrimeraUT_Mesa;


/////////////////////////////////////////////////////////////////////////
/////////////////////////////////////////////////////////////////////////
// ---- Pedir ruta: ...... En Destino
CambioDeMesa_EnDestino_MultiplesGaliboPrimeraUT_Mesa:NOP   0;
      L     21;  // 21 - Generar Evento Pedir Ruta
      T     "DB812_UTs_Control".UT[#NumeroUT].EstadoGeneralUT;
      L     0;  // Dar por tratada
      T     "DB812_UTs_Control".UT[#NumeroUT].EstadoRecepcionUT;

      JU    ContinuarBucleGaliboPrimeraUT_Mesa;


/////////////////////////////////////////////////////////////////////////
/////////////////////////////////////////////////////////////////////////
// ---- Pedir ruta: ...... Sin Destino
CambioDeMesa_SinDestino_MultiplesGaliboPrimeraUT_Mesa:NOP   0;
      L     25;  // 25 - Generar Evento Pedir Ruta (NO DESTINO)
      T     "DB812_UTs_Control".UT[#NumeroUT].EstadoGeneralUT;
      L     0;  // Dar por tratada
      T     "DB812_UTs_Control".UT[#NumeroUT].EstadoRecepcionUT;

      JU    ContinuarBucleGaliboPrimeraUT_Mesa;



/////////////////////////////////////////////////////////////////////////
/////////////////////////////////////////////////////////////////////////
/////////////////////////////////////////////////////////////////////////
// --- (12)- Nueva UT en Mesa
//           * Generar evento
//           * Avisar al generador de ordenes
NuevaEnMesa_MultiplesGaliboPrimeraUT_Mesa:NOP   0;
      L     12;  // 12 - Nueva UT en Mesa
      T     "DB812_UTs_Control".UT[#NumeroUT].EstadoRecepcionUT;
      L     0;  // Darlo por tratado
      T     "DB812_UTs_Control".UT[#NumeroUT].EstadoEmisionUT;

      L     132;  // 132 - Generar Evento de Nueva UT
      T     "DB812_UTs_Control".UT[#NumeroUT].EstadoEventoAGenerar;

      JU    ContinuarBucleGaliboPrimeraUT_Mesa;



NETWORK
TITLE = Tratamiento de Presencia de Bloqueo
// - Ir a la Primera UT de la Mesa
//   * Recoger datos de la UT
//   * Condiciones para tratarla
//   * EstadoEmision Correcto
//     * 0 - Libre
TratarPresenciaBloqueo_Mesa:NOP   0;

/////////////////////////////////////////////////////////////////////////
/////////////////////////////////////////////////////////////////////////
/////////////////////////////////////////////////////////////////////////
// Tratamiento de la Presencia Bloqueo - Primera UT de la Mesa


/////////////////////////////////////////////////////////////////////////
/////////////////////////////////////////////////////////////////////////
// --- Ya se ha encontrado la Primera UT
//     * Recoger datos de la UT
//     * Condiciones de Uso de la Presencia
//       * EstadoRecepcion = 0
//       * EstadoEventosAGenerar = 0
//     * Estado de la Emision Correcto

/////////////////////////////////////////////////////////////////////////
// --- Condiciones de Uso de la Presencia

      L     "DB812_UTs_Control".UT[#NumeroUT].EstadoEventoAGenerar;
      L     0;  // Esta libre
      <>I;  // No se puede hacer nada todavia
      JC    InicioBucle_Mesas;

      L     "DB812_UTs_Control".UT[#NumeroUT].EstadoRecepcionUT;
      L     0;  // Esta libre
      <>I;  // No se puede hacer nada todavia
      JC    InicioBucle_Mesas;


/////////////////////////////////////////////////////////////////////////
// --- Estado de la Emision Correto

      L     "DB812_UTs_Control".UT[#NumeroUT].EstadoEmisionUT;
      L     0;  // 0 - Libre
      <>I;  // No se puede hacer nada todavia
      JC    InicioBucle_Mesas;


/////////////////////////////////////////////////////////////////////////
// --- Generar el Evento
// Jose Antonio Alonso: Modificado 2016 03 21.
//     Poner como Mesa destino la mesa actual.
//     Pero no se elimina la ruta
// Jose Antonio Alonso: Modificado 2020 05 22
//     Activar las Presencias con Bloqueo para multiples UTs

      L     "DB812_UTs_Control".UT[#NumeroUT].Grupo;  // Guardamos el Grupo
      T     #GrupoTMP;

InicioBucleMultiplesUT_PresenciaBloqueo:NOP   0;
      L     122;  // 122 - Generar Evento Peticion de Ruta
      T     "DB812_UTs_Control".UT[#NumeroUT].EstadoEventoAGenerar;
      L     0;  // Darlo por tratado
      T     "DB812_UTs_Control".UT[#NumeroUT].EstadoEmisionUT;

      L     "DB812_UTs_Control".UT[#NumeroUT].MesaActual;  // MesaDestino = MesaActual
      T     "DB812_UTs_Control".UT[#NumeroUT].MesaDestino;

      SET;  // Reset - Memorizar RETI
      R     "DB812_UTs_Control".UT[#NumeroUT].AtributosDeLaUT.MemorizarRETI;


// Comprobar si esta la Mesa Definida como multiples UTs de Salida
      SET;  // Hay que Recorrer el Resto de UTs de la Mesa
      AN    "DB850_DefinicionMesas".Mesa[#NumeroMesa].ConfigMesa.MultiplesCargasDeSalida;
      AN    "DB850_DefinicionMesas".Mesa[#NumeroMesa].ConfigMesa.GrupoDeSalida;
      JC    FinalBucleMultiplesUT_PresenciaBloqueo;

// Hay mas UTs en la Mesa
      L     "DB812_UTs_Control".UT[#NumeroUT].UT_SiguienteMesa;
      T     #SiguienteUT;

      L     #SiguienteUT;
      L     0;
      ==I;  // Hay mas UT's
      JC    FinalBucleMultiplesUT_PresenciaBloqueo;

      L     #SiguienteUT;
      T     #NumeroUT;

// Testear Grupo ?
      SET;
      AN    "DB850_DefinicionMesas".Mesa[#NumeroMesa].ConfigMesa.GrupoDeSalida;
      JC    InicioBucleMultiplesUT_PresenciaBloqueo;

// Dar por tratado solo lo del mismo Grupo
// Grupo Primera UT == Grupo de la Siguiente
      L     "DB812_UTs_Control".UT[#NumeroUT].Grupo;
      L     #GrupoTMP;
      <>I;  // Puede Haber Mas UTs ?
      JC    FinalBucleMultiplesUT_PresenciaBloqueo;
      JU    InicioBucleMultiplesUT_PresenciaBloqueo;


/////////////////////////////////////////////////////////////////////////
// Final del Bucle Multiples UT's en Presencia con Bloqueo
FinalBucleMultiplesUT_PresenciaBloqueo:NOP   0;
      JU    EmpezarProtocolo_Mesa;



NETWORK
TITLE = Tratamiento de Presencia de Reset
// - Todas las UT's de la Mesa
//   No Importa nada: 
//   * Generar Evento 
//   * Incializacion de todo
TratarPresenciaReset_Mesa:NOP   0;

/////////////////////////////////////////////////////////////////////////
/////////////////////////////////////////////////////////////////////////
/////////////////////////////////////////////////////////////////////////

/////////////////////////////////////////////////////////////////////////
// --- Tratamiento de la Presencia Reset - Todas las UT de la Mesa
InicioBuclePresenciaReset_Mesa:NOP   0;

/////////////////////////////////////////////////////////////////////////
// --- Estado de la Emision Correto

      L     "DB812_UTs_Control".UT[#NumeroUT].EstadoEmisionUT;
      L     13;  // Solo en estado 13 (Reset PLC)
      ==I;  // Ir a generar evento del PLC
      JC    Pantalla_PresenciaReset_Mesa;

/////////////////////////////////////////////////////////////////////////
// Ir a generar evento del JdT
      JU    JDT_PresenciaReset_Mesa;

/////////////////////////////////////////////////////////////////////////
// --- Siguinete UT de la Mesa
ContinuarBuclePresenciaReset_Mesa:NOP   0;
      L     "DB812_UTs_Control".UT[#NumeroUT].UT_SiguienteMesa;
      T     #SiguienteUT;

      L     #SiguienteUT;  // ¿Es la Ultima?
      L     0;  // UT Siguiente es 0
      ==I;
      JC    FinPresenciaReset_Mesa;

      L     #SiguienteUT;
      T     #NumeroUT;
      JU    InicioBuclePresenciaReset_Mesa;



/////////////////////////////////////////////////////////////////////////
// --- Fin del Tratamiento de las Presencias de Reset
FinPresenciaReset_Mesa:NOP   0;
// Se ha tratado y hay que cerrar el protocolo
      JU    EmpezarProtocolo_Mesa;



NETWORK
TITLE = ---- Reset Enviado por el JdT
JDT_PresenciaReset_Mesa:NOP   0;

/////////////////////////////////////////////////////////////////////////
/////////////////////////////////////////////////////////////////////////
/////////////////////////////////////////////////////////////////////////
// --- Por cada UT que hay en la Mesa (Reset JdT)
//     * Generar evento
//     * Inicializar las Variables pertinentes


/////////////////////////////////////////////////////////////////////////
// --- No tiene que tener Mckey (NO DEBE DARSE)
      L     "DB812_UTs_Control".UT[#NumeroUT].Mckey;
      L     0;
      <>D;
      JC    ContinuarBuclePresenciaReset_Mesa;

/////////////////////////////////////////////////////////////////////////
// --- Generar Evento
      L     132;  // 132 - Generar Evento de Reset JdT
      T     "DB812_UTs_Control".UT[#NumeroUT].EstadoEventoAGenerar;

      L     0;  // Inicializo
      T     "DB812_UTs_Control".UT[#NumeroUT].EstadoEmisionUT;
      T     "DB812_UTs_Control".UT[#NumeroUT].EstadoRecepcionUT;
      T     "DB812_UTs_Control".UT[#NumeroUT].EstadoGeneralUT;
      T     "DB812_UTs_Control".UT[#NumeroUT].EstadoEventoRecibido;

      JU    ContinuarBuclePresenciaReset_Mesa;



NETWORK
TITLE = ---- Reset Enviado por la Pantalla
Pantalla_PresenciaReset_Mesa:NOP   0;

/////////////////////////////////////////////////////////////////////////
/////////////////////////////////////////////////////////////////////////
/////////////////////////////////////////////////////////////////////////
// --- Por cada UT que hay en la Mesa (Reset PLC)
//     * Generar evento
//     * Inicializar las Variables pertinentes


/////////////////////////////////////////////////////////////////////////
// --- Generar Evento
      L     101;  // 101 - Generar Evento de Reset PLC
      T     "DB812_UTs_Control".UT[#NumeroUT].EstadoEventoAGenerar;
      L     0;  // Inicializo
      T     "DB812_UTs_Control".UT[#NumeroUT].EstadoEmisionUT;
      T     "DB812_UTs_Control".UT[#NumeroUT].EstadoRecepcionUT;
      T     "DB812_UTs_Control".UT[#NumeroUT].EstadoGeneralUT;
      T     "DB812_UTs_Control".UT[#NumeroUT].EstadoEventoRecibido;


/////////////////////////////////////////////////////////////////////////
// --- Control de Memorizacion del Evento RETI
      SET;  // MemoReti Activado
      A     "DB812_UTs_Control".UT[#NumeroUT].AtributosDeLaUT.MemorizarRETI;
      JC    Pantalla_MemorizadoRetirar_PresenciaReset_Mesa;


/////////////////////////////////////////////////////////////////////////
// --- Control de Destino, Hay que Pedir Ruta ....
//     ANULADO 2023 11 >>> No Pedir Ruta >>> Realizar con EstadoRecepcionUT
//      L     "DB812_UTs_Control".UT[#NumeroUT].MesaDestino
//      L     0                    // MesaDestino = 0
//      ==I                        // En Reset
//      SPB   Pantalla_SinDestino_PresenciaReset_Mesa

//      L     "DB812_UTs_Control".UT[#NumeroUT].MesaDestino
//      L     "DB812_UTs_Control".UT[#NumeroUT].MesaActual// MesaDestino = MesaActual
//      ==I                        // En Reset
//      SPB   Pantalla_EnDestino_PresenciaReset_Mesa

/////////////////////////////////////////////////////////////////////////
// Todavia tiene ruta
      L     13;  // Inicializo ?? Reset de la UT
      T     "DB812_UTs_Control".UT[#NumeroUT].EstadoRecepcionUT;

      JU    ContinuarBuclePresenciaReset_Mesa;




/////////////////////////////////////////////////////////////////////////
/////////////////////////////////////////////////////////////////////////
// Pedir Ruta .... En Destino
Pantalla_EnDestino_PresenciaReset_Mesa:NOP   0;
      L     21;  // 21 - Generar Evento Pedir Ruta
      T     "DB812_UTs_Control".UT[#NumeroUT].EstadoGeneralUT;

      JU    ContinuarBuclePresenciaReset_Mesa;


/////////////////////////////////////////////////////////////////////////
/////////////////////////////////////////////////////////////////////////
// Pedir Ruta .... Sin Destino
Pantalla_SinDestino_PresenciaReset_Mesa:NOP   0;
      L     25;  // 25 - Generar Evento Pedir Ruta (NO DESTINO)
      T     "DB812_UTs_Control".UT[#NumeroUT].EstadoGeneralUT;

      JU    ContinuarBuclePresenciaReset_Mesa;


/////////////////////////////////////////////////////////////////////////
/////////////////////////////////////////////////////////////////////////
// Memorizado el Evento RETI
// MesaIntermedia >>> EventoRecibido
Pantalla_MemorizadoRetirar_PresenciaReset_Mesa:NOP   0;
      L     "DB812_UTs_Control".UT[#NumeroUT].MesaIntermedia;
      T     "DB812_UTs_Control".UT[#NumeroUT].EstadoEventoRecibido;

      JU    ContinuarBuclePresenciaReset_Mesa;



NETWORK
TITLE = Tratamiento de Ausencia (NORMAL)
// - Ir a la Primera UT de la Mesa
//   * Recoger datos de la UT
//   * Condiciones para tratarla
//   * EstadoEmision Correcto
//     * 0 - Libre
TratarAusenciaNormal_Mesa:NOP   0;

/////////////////////////////////////////////////////////////////////////
/////////////////////////////////////////////////////////////////////////
/////////////////////////////////////////////////////////////////////////
// Tratamiento de la Ausencia - Primera UT de la Mesa
// Si es Mutiple Ausencia Recorrer toda la Mesa


/////////////////////////////////////////////////////////////////////////
// --- Ya se ha encontrado la Primera UT
//     * Recoger datos de la UT
//     * Condiciones de Uso de la Presencia
//       * EstadoRecepcion = 0
//       * EstadoEventosAGenerar = 0
//     * Estado de la Emision Correcto

/////////////////////////////////////////////////////////////////////////
// --- Condiciones de Uso de la Ausencia

      L     "DB812_UTs_Control".UT[#NumeroUT].EstadoEventoAGenerar;
      L     0;  // Esta libre
      <>I;  // No se puede hacer nada todavia
      JC    FinAusenciaNormal_Mesa;

      L     "DB812_UTs_Control".UT[#NumeroUT].EstadoRecepcionUT;
      L     0;  // Esta libre
      <>I;  // No se puede hacer nada todavia
      JC    FinAusenciaNormal_Mesa;


/////////////////////////////////////////////////////////////////////////
// --- Estado de la Emision Correto

      L     "DB812_UTs_Control".UT[#NumeroUT].EstadoEmisionUT;
      L     0;  // 0 - Libre
      <>I;  // No se puede hacer nada todavia
      JC    FinAusenciaNormal_Mesa;


/////////////////////////////////////////////////////////////////////////
// --- Generar Evento
      L     103;  // 103 - Generar Evento de Ausencia
      T     "DB812_UTs_Control".UT[#NumeroUT].EstadoEventoAGenerar;
      L     0;  // Darlo por tratado
      T     "DB812_UTs_Control".UT[#NumeroUT].EstadoEmisionUT;


/////////////////////////////////////////////////////////////////////////
//     Si Activado Multiples Ausencias recorrer toda la Mesa
      SET;  // Multiples UTs
      AN    "DB850_DefinicionMesas".Mesa[#NumeroMesa].ConfigMesa.AusenciaMultiple;
      JC    EmpezarProtocolo_Mesa;


/////////////////////////////////////////////////////////////////////////
/////////////////////////////////////////////////////////////////////////
/////////////////////////////////////////////////////////////////////////
// --- Generar el Evento de Ausencia para el resto de UT's
// --- Sin condiciones
      L     "DB812_UTs_Control".UT[#NumeroUT].UT_SiguienteMesa;
      T     #SiguienteUT;

InicioBucleAusenciaNormal_Mesa:NOP   0;
      L     #SiguienteUT;
      L     0;
      ==I;
      JC    EmpezarProtocolo_Mesa;

/////////////////////////////////////////////////////////////////////////
// --- Generar Evento
      L     103;  // 103 - Generar Evento de Ausencia
      T     "DB812_UTs_Control".UT[#SiguienteUT].EstadoEventoAGenerar;
      L     0;  // Darlo por tratado
      T     "DB812_UTs_Control".UT[#SiguienteUT].EstadoEmisionUT;


/////////////////////////////////////////////////////////////////////////
// --- Siguiente UT de la Mesa
      L     "DB812_UTs_Control".UT[#SiguienteUT].UT_SiguienteMesa;
      T     #SiguienteUT;

      JU    InicioBucleAusenciaNormal_Mesa;


/////////////////////////////////////////////////////////////////////////
// --- Fin del Tratamiento de las Ausencias
FinAusenciaNormal_Mesa:NOP   0;
// No se ha tratado la Ausencia
      JU    InicioBucle_Mesas;



NETWORK
TITLE = Tratamiento de Ausencia (BORRAR UT)
// - Ir a la Primera UT de la Mesa
//   * Recoger datos de la UT
//   * Condiciones para tratarla
//   * EstadoEmision Correcto
//     * 0 - Libre
TratarAusenciaBorrar_Mesa:NOP   0;

/////////////////////////////////////////////////////////////////////////
/////////////////////////////////////////////////////////////////////////
/////////////////////////////////////////////////////////////////////////
// Tratamiento de la Ausencia - Primera UT de la Mesa
// Si es Mutiple Ausencia Recorrer toda la Mesa


/////////////////////////////////////////////////////////////////////////
// --- Ya se ha encontrado la Primera UT
//     * Recoger datos de la UT
//     * Condiciones de Uso de la Presencia
//       * EstadoRecepcion = 0
//       * EstadoEventosAGenerar = 0
//     * Estado de la Emision Correcto


/////////////////////////////////////////////////////////////////////////
// --- Condiciones de Uso de la Ausencia

      L     "DB812_UTs_Control".UT[#NumeroUT].EstadoEventoAGenerar;
      L     0;  // Esta libre
      <>I;  // No se puede hacer nada todavia
      JC    FinAusenciaBorrar_Mesa;

      L     "DB812_UTs_Control".UT[#NumeroUT].EstadoRecepcionUT;
      L     0;  // Esta libre
      <>I;  // No se puede hacer nada todavia
      JC    FinAusenciaBorrar_Mesa;


/////////////////////////////////////////////////////////////////////////
// --- Estado de la Emision Correto

      L     "DB812_UTs_Control".UT[#NumeroUT].EstadoEmisionUT;
      L     0;  // 0 - Libre
      <>I;  // No se puede hacer nada todavia
      JC    FinAusenciaBorrar_Mesa;


/////////////////////////////////////////////////////////////////////////
// --- Generar Evento
      L     131;  // 131 - Generar Evento de Borrar UT
      T     "DB812_UTs_Control".UT[#NumeroUT].EstadoEventoAGenerar;
      L     0;  // Darlo por tratado
      T     "DB812_UTs_Control".UT[#NumeroUT].EstadoEmisionUT;


/////////////////////////////////////////////////////////////////////////
//     Si Activado Multiples Ausencias recorrer toda la Mesa
      SET;  // Multiples UTs
      AN    "DB850_DefinicionMesas".Mesa[#NumeroMesa].ConfigMesa.AusenciaMultiple;
      JC    EmpezarProtocolo_Mesa;


/////////////////////////////////////////////////////////////////////////
/////////////////////////////////////////////////////////////////////////
/////////////////////////////////////////////////////////////////////////
// --- Generar el Evento de Ausencia para el resto de UT's
// --- Sin condiciones
      L     "DB812_UTs_Control".UT[#NumeroUT].UT_SiguienteMesa;
      T     #SiguienteUT;

InicioBucleAusenciaBorrar_Mesa:NOP   0;
      L     #SiguienteUT;
      L     0;
      ==I;
      JC    EmpezarProtocolo_Mesa;

/////////////////////////////////////////////////////////////////////////
// --- Generar Evento
      L     131;  // 131 - Generar Evento de Borrar UT
      T     "DB812_UTs_Control".UT[#SiguienteUT].EstadoEventoAGenerar;
      L     0;  // Darlo por tratado
      T     "DB812_UTs_Control".UT[#SiguienteUT].EstadoEmisionUT;


/////////////////////////////////////////////////////////////////////////
// --- Siguiente UT de la Mesa
      L     "DB812_UTs_Control".UT[#SiguienteUT].UT_SiguienteMesa;
      T     #SiguienteUT;

      JU    InicioBucleAusenciaBorrar_Mesa;


/////////////////////////////////////////////////////////////////////////
// --- Fin del Tratamiento de las Ausencias
FinAusenciaBorrar_Mesa:NOP   0;
// No se ha tratado la Ausencia
      JU    InicioBucle_Mesas;



NETWORK
TITLE = Finalizar la funcion
// Se acabo la funcion

_END: NOP   0;

END_FUNCTION
